VAR_GLOBAL CONSTANT
	iMAX_AXES_REF : INT := 5;
END_VAR
VAR_GLOBAL
	iGlobalCounter : UINT;
	fbCrititcalSection : FB_IecCriticalSection;
END_VAR

(* stored: Version 1.1.0.1, ProductVersion 3.1.4024.11
   GVL GVL: Id {b31223e4-d801-463b-aea4-2814692ede38} *)
